// TIA Portal V21 export
VAR_GLOBAL   // PLC tag table "K_Motore_Filler"
END_VAR
VAR_GLOBAL CONSTANT   // user constants
   K_Motore_Filler_Volume : Int := 0;
END_VAR
